(* Logix 5000 project; controller Counters Emulate 5570 rev 33.11; software revision 33.00 *)

TASK T00_MainTask (continuous, watchdog 500 ms) : P00_MainProgram

MODULES
   Local : Emulate 5570 (ICP 2, rev 33.11)
END_MODULES

PROGRAM P00_MainProgram   (* main routine R00_MainRoutine *)
VAR
   Counter : COUNTER;
END_VAR

ROUTINE R00_MainRoutine   (* ladder *)
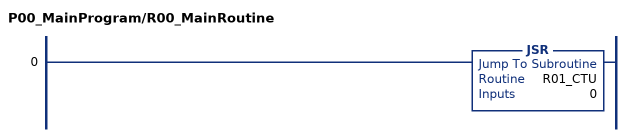
   0: JSR(R01_CTU,0);
END_ROUTINE

ROUTINE R01_CTU   (* ladder *)
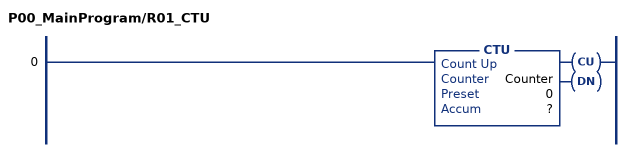
   0: CTU(Counter,?,?);
END_ROUTINE
END_PROGRAM
